Universal Robots PolyScope program: socket_sample.urp

Program socket_sample (installation=default directory=/home/ur/ursim-current/programs createdIn=5.6.0.90886 lastSavedIn=5.6.0.90886 robotSerialNumber=20195699999)
Calibrated DH parameters: a=[0, -0.4784, -0.36, 0, 0, 0]; d=[0.1807, 0, 0, 0.17415, 0.11985, 0.11655]; alpha=[1.570796, 0, 0, 1.570796, -1.570796, 0]; deltaTheta=[0, 0, 0, 0, 0, 0]
Robot Program (runOnlyOnce=true)
  Script: socket_open("192.168.0.5", 50001)
  Script: socket_open("192.168.0.5", 50001,"socket_custom")
  Script: socket_send_string("Hello from socket !")
  Wait Sleep waitTime=1
  a := socket_get_var("var_a")
  Wait Sleep waitTime=1
  Script: socket_close()
  str := socket_read_string("socket_custom", timeout=10)
  Script: socket_close("socket_custom")
